//****************************************************************************************************
// Code generated by SFC Generator V1.13 on 13/03/19 15:52:14 by  David Paspa from File G:\Business\Synertec\MPI.SMS\automation\code\awlMaster\stencil\seq_hdr.awl
//****************************************************************************************************
//****************************************************************************************************

//================================ SEQ HEADER ================================//
//            Copyright 2018 Rieckermann Engineering Operations               //
//----------------------------------------------------------------------------//
// Title: PH_EMX1_SETUP_FILTER                                                       //
//                                                                            //
// Description:                                                               //
// Setup MMFLx for Filtration                                                        //
//                                                                            //
// // SFC Revision History:
// Rev By               Date        CC         Note
// 2.0 David Paspa      27-Nov-2018            Reboot for S7-1500
// 0.4 Khairul Basar    07-Sep-2009 CC-09/023  Prompt_filter is reset in Step2.
// 0.3 Khairul Basar    25-Aug-2009 CC-09/023  Change in Verific,& TRN code OR to AND
//                                             Change in the Last step.
// 0.2 Khairul Basar    18-Aug-2009            Added logic code
// 0.1 David Paspa      13-Jul-2009            SFC structural design                                                       //
//----------------------------------------------------------------------------//
// Sequencer Revision History:                                                //
// Rev By               Date        CC        Note                            //
// 2.0 David Paspa      05-Jan-2018 NA        Reboot for S7-1500.             //
// 1.6 Khairul Basar    19-Nov-2009 NA        Reset #sqSequencer.STEP.Active  //
//                                            when STEP Finished.             //
// 1.5 Khairul Basar    15-Oct-2009 NA        Placeholder inserted:           //
//                                            "udtSQ_PH";          //
// 1.4 Khairul Basar    06-Oct-2009 NA        R #PAUSE;                       //
// 1.3 Khairul Basar    30-Sep-2009 NA        SEQ_HDR change STEP-0 code      //
//                                            deleted.                        //
// 1.2 Khairul Basar    26-Sep-2009 NA        Refer R4.                       //
// 1.1 Khairul Basar    23-Sep-2009 NA        Refer R3.                       //
// 1.0 Khairul Basar    20-Sep-2009 NA        STEP.Finished flag reset by     //
//                                            JUMP_MAN.                       //
// 0.9 Khairul Basar    11-Sep-2009 NA        SQ_TIMER added as VAR, declared //
//                                            in SEQ_FTR.                     //
// 0.8 Khairul Basar    09-Sep-2009 NA        SqSequencer.Err_Fault is reset  //
//                                            on Stop cmd, Step-0 dead code   //
//                                            deleted from ACT & Verify.      //
//                                            STP_FTR Step_withErr flag       //
//                                            STEP_NUM place holder           //
//                                            configured.                     //
// 0.7 Khairul Basar    28-Aug-2009 NA        SQ_FINISHED OUT added again.    //
//                                            Deleted during major mod R3.    //
// 0.6 Khairul Basar    23-Aug-2009 NA        Refer R2.                       //
// 0.5 Khairul Basar    23-Aug-2009 NA        Refer R1.                       //
// 0.4 Khairul Basar    18-Aug-2009 NA        Reset Step done with/out error  //
//                                            bits using FC:RSET.             //
// 0.3 David Paspa      16-Aug-2009 NA        Added placeholders for header   //
//                                            name and version and revision   //
//                                            history.                        //
// 0.2 Khairul Basar    11-Aug-2009 NA        Retired external udt file for   //
//                                            Static type parameters. All     //
//                                            parameters now IN, OUT or       //
//                                            IN_OUT.                         //
// 0.1 Khairul Basar    12-Jun-2009 NA        Initial design.                 //
//----------------------------------------------------------------------------//
// R4:                                                                        //
// 1.If SQ not finished Resume command will start Step timer, and redo the    //
// last action, verify the feedback.                                          //
// 2."STEP.finished" flag is ANDed with "TRN_AND_JUMP" in the snippet file    //
// TRN_HDR.This is to avoid checking of transition logic if STEP is not       //
// finished yet.                                                              //
// 3.MDCH, Load & transfer typo corrected.                                    //
//                                                                            //
// R3:                                                                        //
// 1.SqStepTimer.IN is reset in STEP_FTR instead of resetting it in TRN_HDR.  //
// This is because TRN_HDTR is not included in the Last step and StepTimer    //
// must reset in the last step.                                               //
// 2.Reset all the timers when SQ stops.Reset done in SEQ_HDR.                //
// Also STEP-finished flag reset when SQ is OFF to                            //
// scan last step.                                                            //
//                                                                            //
// R2:                                                                        //
// 1.Any step error will send the Sequencer into Pause state.Code added in    //
// SEQ_HDR.Snippet Place holder for Bool-array 8 is   //
// deleted.                                                                   //
//                                                                            //
// R1:                                                                        //
// 1.sqStepTimer:All Verification Code must satisfy the condition finish step //
// action within STEP_DELAY time(40s).If step actions not finished within the //
// time period the error flag will raise High signal.Else timer will reset.   //
// 2.sqRunTimer Added therefore can be used as retentive & non retentive.     //
// 3.sqSequencer: This is re-structured UDT which is redefined the symbol     //
// names as well as it gives more clearity.                                   //
// 4.fcMODE and fcCMD functions are added to handle the mode & command        //
// independently regardless of other logic.Two separate UDT udtMODE & udt     //
// CMD assigned to Mode & command function respectively.                      //
// 5.MAN_JUMP programed for manual mode jump operation with or without        //
// Transition code satisfied.TRN_AND_JUMP & NO_VERIFC are the parameters      //
// which will define whether verification code & transition code need to be   //
// checked to perform jump operation.                                         //
// 6.Auto to Manual switchover will be bumpless & will not affect step        //
// operation.Manual to auto switchover can be used to resume Step action at   //
// defined.                                                                   //
// Step number entered in STEPNO_JUMP.                                        //
//                                                                            //
// Parameters:                                                                //
// INPUTS                                                                     //
// ======                                                                     //
// SQ_CMD          Sequence command input inherited from object block         //
//                 0: off/idle                                                //
//                 1: start/initiate                                          //
//                 2: pause                                                   //
//                 3: resume                                                  //
//                 4: reserved (not programmed)                               //
//                 5: reserved (not programmed)                               //
//                 6: abort/go to last step                                   //
//                 7: acknowledge error/fault                                 //
// SQ_MODE         Sequencer Auto/Manual input inherited from object block    //
//                 1: manual                                                  //
//                 2: auto                                                    //
//                                                                            //
// INPUT/OUTPUTS                                                              //
// =============                                                              //
// SQ_JUMP_MAN     Allows manual jumping from one step to the next step. The  //
//                 manual jump flag is ORed with the transition process       //
//                 condition and so can be used to bypass the condition if the//
//                 sequence will not progress.                                //
//                 This input can also be used to jump to any step even       //
//                 when no transition -> step linkage exists. This is only    //
//                 possible when the SQ_MODE is in manual and SQ is in the    //
//                 idle step. The step to jump to is specified in             //
//                 SQ_man_jump_to_step (not accesseble by this FB in/out      //
//                 interface but a separate DB memory location).              //
//                                                                            //
// OUTPUTS                                                                    //
// =======                                                                    //
// SQ_STATE        The calculated state of the sequence                       //
//                 0: off/idle                                                //
//                 1: start/initiated                                         //
//                 2: paused                                                  //
//                 3: resumed                                                 //
//                 4: reserved (wrong Mode)                                   //
//                 5: reserved (Wrong commad)                                 //
//                 6: aborted/go to last step                                 //
//                 7: acknowledged error/fault                                //
// CURSTEP         Current step being proccessed.                             //
// S_ACTIVE        If current step is active                                  //
// NXT_STEP        Next step to jump to if transition condition is true       //
// ERR_FAULT       True if any error/ or fault present                        //
// PAUSED          True if step is paused                                     //
// OFF_IDLE        Sequence is not running but ready for next SQ (in step=0)  //
//----------------------------------------------------------------------------//
// Define variables:                                                          //
//----------------------------------------------------------------------------//
FUNCTION_BLOCK "fbPH_EMX1_SETUP_FILTER"
TITLE = PH : EMX1_SETUP_FILTER
{ S7_Optimized_Access := 'TRUE' }
NAME : X1_FILT
AUTHOR : REO
VERSION : 2.0

VAR_IN_OUT
    _zsc_filter_state :INT ;	//MMFLx Filter connection sensor switch.

    _zsc_filter_cmd :INT ;	//FILTER connection command
    _zsc_cipsip_cmd :INT ;	//CIPSIP connection command


    dummy : bool;            // Dummy placeholder for call without comma
END_VAR

VAR
    smc : "udtModeCommandSFC";         // SFC mode and command
    sqStepTimer : "TON";
    sqRunTimer : "fbRunTimer";
    sqSequencer : "udtSFCSequence32";
    SQ_TIMER: "TON";
    SQ_TIMER2: "TON";
    SQ_TIMER3: "TON";
    sqSeqTimerStart : Bool;
    sqSeqTimerStart2 : Bool;
    sqSeqTimerStart3 : Bool;
    sqSeqTimerElapsed : Time;
    sqSeqTimerElapsed2 : Time;
    sqSeqTimerElapsed3 : Time;
    sqSeqTimerExpired : Bool;
    sqSeqTimerExpired2 : Bool;
    sqSeqTimerExpired3 : Bool;
    sqStepTimerElapsed : Time;
    sqStepTimerExpired : Bool;
    _log_msg_confirm_connect :BOOL ;	//PH_EMX1_SETUP_FILTER OPerator to confirm filters connected confirmed yes
    _log_msg_setup_filter_begin :BOOL ;	//PH_EMX1_SETUP_FILTER begin time
    _log_msg_setup_filter_end :BOOL ;	//PH_EMX1_SETUP_FILTER end time
    _prompt_connect_filter_confirm_yes :BOOL ;	//PH_EMX1_SETUP_FILTER operator to confirm filters connected confirmed yes
    _prompt_connect_filter :BOOL ;	//PH_EMX1_SETUP_FILTER Operator to confirm filters connected

END_VAR

BEGIN
NETWORK
TITLE =Call Mode checking function
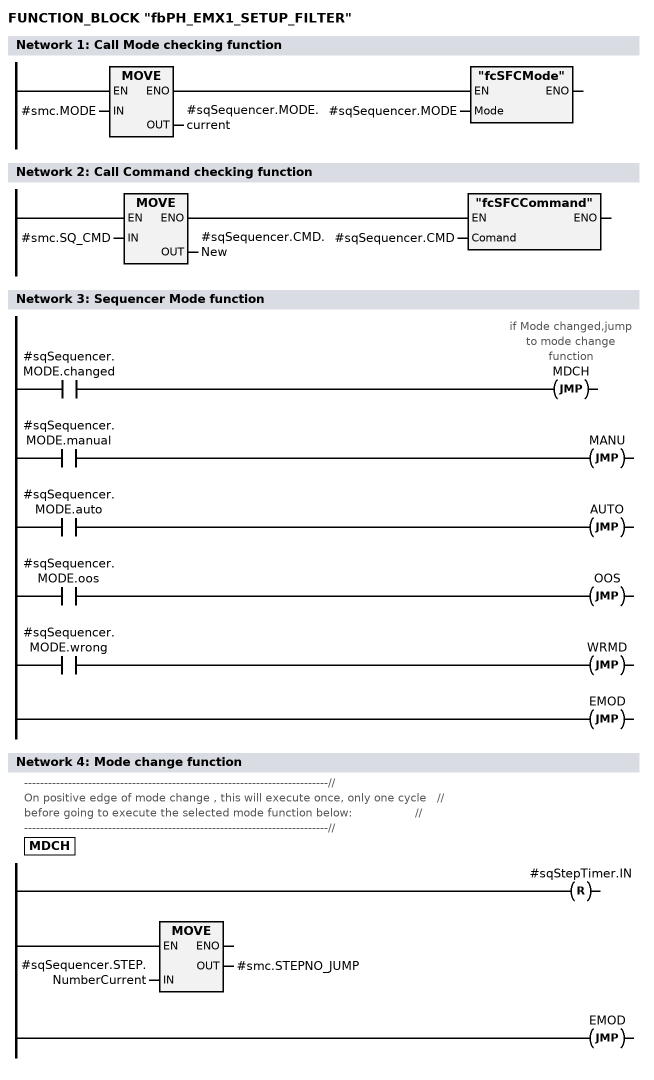
    L     #smc.MODE;
    T     #sqSequencer.MODE.current;
    CALL "fcSFCMode"
    (   Mode                 := #sqSequencer.MODE
    );

NETWORK
TITLE =Call Command checking function
    L     #smc.SQ_CMD;
    T     #sqSequencer.CMD.New;
    CALL "fcSFCCommand"
    (   Comand               := #sqSequencer.CMD
    );

NETWORK
TITLE =Sequencer Mode function

      A     #sqSequencer.MODE.changed;
      JC    MDCH; // if Mode changed,jump to mode change function
      A     #sqSequencer.MODE.manual;
      JC    MANU;
      A     #sqSequencer.MODE.auto;
      JC    AUTO;
      A     #sqSequencer.MODE.oos;
      JC    OOS;
      A     #sqSequencer.MODE.wrong;
      JC    WRMD;
      JU    EMOD;

NETWORK
TITLE =Mode change function
//----------------------------------------------------------------------------//
// On positive edge of mode change , this will execute once, only one cycle   //
// before going to execute the selected mode function below:                  //
//----------------------------------------------------------------------------//
MDCH: NOP   0;
      SET   ;
      R     #sqStepTimer.IN;
      L     #sqSequencer.STEP.NumberCurrent;
      T     #smc.STEPNO_JUMP;
      JU    EMOD;

NETWORK
TITLE =Manual Mode function
//----------------------------------------------------------------------------//
// #TRN_AND_JUMP=can set/reset                                                //
// #sqSequencer.STEP.JumpCtrl=Can set/reset by #MAN_JUMP                      //
// #NO_VERIFIC=Can set/ Reset                                                 //
//----------------------------------------------------------------------------//
MANU: NOP   0; //Manual mode selected



      A     #smc.MAN_JUMP;
      =     #sqSequencer.STEP.JumpCtrl;
      A     #smc.MAN_JUMP;
      JCN   EMOD;

      L     #smc.STEPNO_JUMP;
      T     #sqSequencer.STEP.NumberNext;
      T     #sqSequencer.STEP.NumberCurrent;
      R     #smc.MAN_JUMP; //Reset MAN_JUMP after loading user destination Step number
      R     #sqSequencer.STEP.Finished; //Reset finish flag, to execute next step action
      JU    EMOD;

NETWORK
TITLE =Auto Mode function
//----------------------------------------------------------------------------//
// #TRN_AND_JUMP=always set                                                   //
// #sqSequencer.STEP.JumpCtrl=Always set                                      //
// #NO_VERIFIC=Alwasy Reset                                                   //
//----------------------------------------------------------------------------//
AUTO: NOP   0; //Auto mode selected



      R     #smc.MAN_JUMP;
      S     #smc.TRN_AND_JUMP;
      R     #smc.NO_VERIFIC;
      S     #sqSequencer.STEP.JumpCtrl; //Always Set in auto mode

      L     #sqSequencer.STEP.NumberCurrent;
      T     #smc.STEPNO_JUMP;
      JU    EMOD;
NETWORK
TITLE =OOS mode function

OOS:  NOP   0; // Out of service
      JU    EMOD;
WRMD: NOP   0; //Wrong mode selected
      S     #sqSequencer.Error_Fault;
      L     "dbCONST".SEQ.STATE.WRMODE;
      T     #smc.SQ_STATE;

      JU    EMOD;

NETWORK
TITLE =Mode not changedd

      NOP   0;

NETWORK
TITLE =End Mode function

EMOD: NOP   0;

NETWORK
TITLE =An error will Pause the Sequencer,Operator must Resume SQ to run

      A     #sqSequencer.Error_Fault;
      AN    #sqSequencer.CMD.Changed;
      JC    PAUS;

NETWORK
TITLE =Command Action function

      A     #sqSequencer.CMD.Changed;
      JCN   CNCH; // if Command not changed,jump to end function
      R     #sqStepTimer.IN;

      A     #sqSequencer.CMD.Start;
      JC    STRT;

      A     #sqSequencer.CMD.Stop;
      JC    STOP;

      A     #sqSequencer.CMD.Pause;
      JC    PAUS;

      A     #sqSequencer.CMD.Resume;
      JC    RESM;

      A     #sqSequencer.CMD.Abort;
      JC    _abrt_begin;

      A     #sqSequencer.CMD.Ack;
      JC    ACKN;

      A     #sqSequencer.CMD.wrong;
      JC    WCMD;

      JU    ECMD; //Wrong command/not specified command
//End Comand function

NETWORK
TITLE =Comand -Start/Initiate action function

STRT: NOP   0;
      R     #smc.OFF_IDLE;
      R     #smc.ABORTED;
      R     #smc.PAUSED;
      R     #sqSequencer.STEP.Active;
      R     #sqSequencer.STEP.Finished;
      R     #sqSequencer.STEP.ActionFinished;
      R     #sqSequencer.STEP.Jump;
      R     #sqSequencer.STEP.TimerExpired;
      R     #sqSequencer.STEP.Error_Fault;
      R     #sqSequencer.STEP.ActionVerified;
      R     #sqStepTimer.IN;

//      S     #sqRunTimer.RESET;

//----------------------------------------------------------------------------//
// Load Initial step Number:                                                  //
//----------------------------------------------------------------------------//
      L     1;
      T     #sqSequencer.STEP.Initial;
      L     #sqSequencer.STEP.Initial;
      T     #sqSequencer.STEP.NumberCurrent;
      T     #sqSequencer.STEP.NumberNext;

      L     "dbCONST".SEQ.STATE.STARTED;
      T     #smc.SQ_STATE;

NETWORK
TITLE = Reset sequence Done bits
    //------------------------------------------------------------------------//
    // Reset Step done bits:                                                  //
    //------------------------------------------------------------------------//
    CALL FILL_BLK
    {value_type := 'Bool', count_type := 'UInt'}
    (   IN                   := 0 ,
        COUNT                := 32 ,
        OUT                  := #sqSequencer.STEP.Done[1]
    );

NETWORK
TITLE = Reset sequence Error bits
    //------------------------------------------------------------------------//
    // Reset Step error bits:                                                 //
    //------------------------------------------------------------------------//
    CALL FILL_BLK
    {value_type := 'Bool', count_type := 'UInt'}
    (   IN                   := 0 ,
        COUNT                := 32 ,
        OUT                  := #sqSequencer.STEP.WithError[1]
    );

    JU    ECMD; //End Function

NETWORK
TITLE =Comand -Stop action function

STOP: NOP   0;
      S     #smc.OFF_IDLE;
      R     #sqSequencer.STEP.Active;
      R     #sqSequencer.STEP.Finished;
      R     #sqSequencer.STEP.ActionFinished;
      R     #sqSequencer.STEP.Jump;
      R     #sqSequencer.STEP.TimerExpired;
      R     #sqSequencer.STEP.Error_Fault;
      R     #sqSequencer.Error_Fault;
      R     #sqSequencer.STEP.ActionVerified;
      R     #sqRunTimer.ENABLE;
      R     #sqStepTimer.IN;
      R     #sqSeqTimerStart;
      R     #sqSeqTimerStart2;
      R     #sqSeqTimerStart3;
      R     #smc.PAUSED;
      R     #smc.ABORTED;


//Go to last step
      L     4;
      T     #sqSequencer.FinalStep;
      T     #sqSequencer.STEP.NumberNext;

      JU    ECMD; //End Function

NETWORK
TITLE =Comand -Pause action function

PAUS: NOP   0;
      S     #smc.PAUSED;
      R     #smc.S_ACTIVE;
      S     #sqRunTimer.PAUSE;
      L     #sqSequencer.STEP.NumberCurrent;
      T     #smc.STEPNO_JUMP;
      L     "dbCONST".SEQ.STATE.PAUSED;
      T     #smc.SQ_STATE;

      JU    ECMD; //End Function

NETWORK
TITLE =Comand -Resume action function

RESM: NOP   0;
      R     #smc.PAUSED;
      R     #sqRunTimer.PAUSE;
      R     #sqStepTimer.IN; //Reset Step timer
      L     "dbCONST".SEQ.STATE.RESUMED;
      T     #smc.SQ_STATE;

      A     #smc.SQ_FINISHED;
      JC    ECMD;
      R     #sqSequencer.STEP.Active;
      R     #sqSequencer.STEP.Finished;
      R     #sqSequencer.STEP.ActionFinished;

      JU    ECMD; //End Function

NETWORK
TITLE =Comand -Abort action function

_abrt_begin: NOP   0;

      S     #smc.ABORTED;
      R     #sqSequencer.STEP.Active;
      R     #sqSequencer.STEP.Finished;
      R     #sqSequencer.STEP.ActionFinished;
      R     #sqSequencer.STEP.Jump;
      R     #sqSequencer.STEP.TimerExpired;
      R     #sqSequencer.STEP.Error_Fault;
      R     #sqSequencer.Error_Fault;
      R     #sqSequencer.STEP.ActionVerified;
      R     #sqRunTimer.ENABLE;
      R     #sqStepTimer.IN;
      R     #sqSeqTimerStart;
      R     #sqSeqTimerStart2;
      R     #sqSeqTimerStart3;
      R     #smc.PAUSED;
      R     #smc.OFF_IDLE;


//Go to last step
      L     4;
      T     #sqSequencer.FinalStep;
      T     #sqSequencer.STEP.NumberNext;

      JU    ECMD;

NETWORK
TITLE =Comand -Acknowledge action function

ACKN: NOP   0;
      R     #smc.ERR_FAULT;
      R     #sqSequencer.Error_Fault;
      L     "dbCONST".SEQ.STATE.ACKNOWLEDGED;
      T     #smc.SQ_STATE;

      JU    ECMD; //End Function

NETWORK
TITLE =Comand -wrong/unavailable

WCMD: NOP   0;

      S     #sqSequencer.Error_Fault;
      L     "dbCONST".SEQ.STATE.WRCMD;
      T     #smc.SQ_STATE;

      JU    ECMD;
NETWORK
TITLE =Comand -not changedd

CNCH: NOP   0; // Command not changed

NETWORK
TITLE =End command Function

ECMD: NOP   0;

NETWORK
TITLE =Sequencer Step Jump distrubution list
    //------------------------------------------------------------------------//
    // Sequencer step jump list. Load the step number to execute the step:    //
    //------------------------------------------------------------------------//
    L     #sqSequencer.STEP.NumberCurrent;
    JL    SQER; // If Sequencer Step number invalid or greater than available number of step
    JU    S000; // Exceptional Error Handling
    JU    S001; // STEP-001:
JU    S002; // STEP-002:
JU    S003; // STEP-003:
JU    S004; // STEP-004:


    //------------------------------------------------------------------------//
    // If Step number is Invalid or Out of Range:                             //
    //------------------------------------------------------------------------//
SQER: NOP   0;
    A     "alwaysLow";
    S     #sqSequencer.Error_Fault;
    JU    COMM; // Jump to Common Sequencer code handling function

NETWORK
TITLE =STEP0 STEP0 STEP0 STEP0 STEP0 STEP0 STEP0 STEP0 STEP0 STEP0 STEP
    //------------------------------------------------------------------------//
    // STEP0 STEP0 STEP0 STEP0 STEP0 STEP0 STEP0 STEP0 STEP0 STEP0 STEP0 STEP //
    // AUTOCODE   AUTOCODE   AUTOCODE   AUTOCODE   AUTOCODE   AUTOCODE   AUTO //
    // STEP0 STEP0 STEP0 STEP0 STEP0 STEP0 STEP0 STEP0 STEP0 STEP0 STEP0 STEP //
    //------------------------------------------------------------------------//

NETWORK
TITLE =S000: STEP0::If Paused exit

S000: NOP   0;
      JU    COMM;






NETWORK
TITLE =S001: STEP-01::PH_EMX1_SETUP_FILTER : SETUP CIPSIP begin.
    //================================ STEP HEADER ===========================//
    // STEP001 STEP001 STEP001 STEP001
    // AUTOCODE   AUTOCODE   AUTOCODE   AUTOCODE   AUTOCODE   AUTOCODE   AUTO //
    // STEP001 STEP001 STEP001 STEP001
    //------------------------------------------------------------------------//
    // Log SETUP FILTER begin time.
    //------------------------------------------------------------------------//
S001: NOP   0;

      SET;
      R     #sqSequencer.STEP.jumpDone[01];
      A     #sqSequencer.CMD.Pause; //If paused jump
      JC    COMM;

NETWORK
TITLE =S001:STEP-01:Begin Action

      A     #sqSequencer.STEP.Finished;
      JC    A001; // Exit Action code, Jump to A001 Transition code

      //----------------------------------------------------------------------//
      // Begin step Action:                                                   //
      //----------------------------------------------------------------------//
      A     #sqSequencer.STEP.Active;
      JC    L001; // Action number loaded, Jump to L001--Step Action List

      //----------------------------------------------------------------------//
      // Load Default/Initial Step action number:                             //
      //----------------------------------------------------------------------//
      S     #sqSequencer.STEP.Active;
      S     #sqStepTimer.IN;
      L     1; //First Action, Step must contain Minimum one action
      T     #sqSequencer.STEP.ActionNumber;

//----------------------------------------------------------------------------//
// Step action list.                                                          //
// aann=mini Action step number(aa) inside main step number(nn)               //
// First Action aa00, Second action ab00, Third ac00, etc.                    //
//----------------------------------------------------------------------------//
L001: NOP   0;

      L     #sqSequencer.STEP.ActionNumber;
      JL    r001; //Wrong Action number
      JU    _001; //Action error handling
       JU    aa01; //ACTION-01


//----------------------------------------------------------------------------//
// More step action in the list can be inserted here, upto ab is tested:      //
//----------------------------------------------------------------------------//
r001: NOP   0; //Wrong action number
      S     #sqSequencer.Error_Fault;
      JU    k001; //Exit
_001: NOP   0; // Action error handling
      JU    k001; // Exit






NETWORK
TITLE =S001:: STEP-001:: : ACTION CODE
    //================================ ACT HEADER ============================//
    // ACTION ACTION ACTION ACTION ACTION ACTION ACTION ACTION ACTION ACTION  //
    // AUTOCODE   AUTOCODE   AUTOCODE   AUTOCODE   AUTOCODE   AUTOCODE   AUTO //
    // ACTION ACTION ACTION ACTION ACTION ACTION ACTION ACTION ACTION ACTION  //
    //------------------------------------------------------------------------//
    // //Log SETUP FILTER begin time.
    aa01: NOP   0;

    //------------------------------------------------------------------------//
    // ACT ACT ACT ACT ACT ACT ACT ACT ACT ACT ACT ACT ACT ACT ACT ACT ACT    //
    //------------------------------------------------------------------------//
    //Log SETUP FILTER begin time.
SET;
S #_log_msg_setup_filter_begin;

// Send IN command to FILTER zsc.
L "dbCONST".BLK.ZSC2.CMD.IN;
T  #_zsc_filter_cmd;

// Send OUT command to CIPSIP zsc.
L "dbCONST".BLK.ZSC2.CMD.OUT;
T #_zsc_cipsip_cmd;

    //------------------------------------------------------------------------//
    // VERIFY  VERIFY VERIFY VERIFY VERIFY VERIFY VERIFY VERIFY VERIFY VERIFY //
    //------------------------------------------------------------------------//
    A "uncondJump";
    S     #sqSequencer.STEP.ActionVerified; //Action verified

    //------------------------------------------------------------------------//
    // Action done:                                                           //
    //------------------------------------------------------------------------//
    O     #sqSequencer.STEP.ActionVerified;
    O     #smc.NO_VERIFIC;       //No verification , bypass verification code
    S     #sqSequencer.STEP.ActionFinished;






    //============================= STEP FOOTER ==============================//
    // AUTOCODE   AUTOCODE   AUTOCODE   AUTOCODE   AUTOCODE   AUTOCODE   AUTO //
    // Get Ready after action finished:                                       //
    //------------------------------------------------------------------------//
    A     #sqSequencer.STEP.ActionFinished;
    JCN   k001;

    //------------------------------------------------------------------------//
    // Reset Action finished flag, ready for next step action:                //
    //------------------------------------------------------------------------//
    R     #sqSequencer.STEP.ActionVerified;
    R     #sqSequencer.STEP.ActionFinished;

    //------------------------------------------------------------------------//
    // If ALL actions are finished:                                           //
    //------------------------------------------------------------------------//
    SET   ;
    S     #sqSequencer.STEP.Finished;
    R     #sqSequencer.STEP.Active;
    S     #sqSequencer.STEP.Done[01];

    //------------------------------------------------------------------------//
    // End Step action(s):                                                    //
    //------------------------------------------------------------------------//
    JU    k001;

//----------------------------------------------------------------------------//
// Finished Step Action(s):                                                   //
//----------------------------------------------------------------------------//
k001: NOP   0;

    A     #sqStepTimerExpired;
    S     #sqSequencer.STEP.WithError[01]; // Step error flag
    S     #sqSequencer.Error_Fault;
    R     #sqStepTimer.IN;

NETWORK
TITLE =S001:STEP-001::Begin Transition
    //------------------------------------------------------------------------//
    // Begin the transition code:                                             //
    //------------------------------------------------------------------------//
    A001: NOP   0;
    R     #sqStepTimer.IN;






    //============================= TRAN HEADER ==============================//
    // AUTOCODE   AUTOCODE   AUTOCODE   AUTOCODE   AUTOCODE   AUTOCODE   AUTO //
    // Bypass transition if manual jump:                                      //
    //------------------------------------------------------------------------//
    A     #sqSequencer.STEP.Finished;
    A     #smc.TRN_AND_JUMP;     //Manual jump is set Transition as bypassed
    JCN   COMM;              //exit

NETWORK
TITLE =S001::STEP 001:TRAN 001: Unconditional Jump
//----------------------------------------------------------------------------//
// TRAN   TRAN   TRAN   TRAN   TRAN   TRAN   TRAN   TRAN   TRAN   TRAN   TRAN //
// TRAN   TRAN   TRAN   TRAN   TRAN   TRAN   TRAN   TRAN   TRAN   TRAN   TRAN //
//----------------------------------------------------------------------------//
// Jump
//----------------------------------------------------------------------------//
// CONDITION   CONDITION   CONDITION   CONDITION   CONDITION   CONDITION   CO //
// CONDITION   CONDITION   CONDITION   CONDITION   CONDITION   CONDITION   CO //
//----------------------------------------------------------------------------//
A "uncondJump";






    //============================= TRAN FOOTER ==============================//
    // Transition jump control:                                               //
    //------------------------------------------------------------------------//
    A     #sqSequencer.STEP.JumpCtrl;
    S     #sqSequencer.STEP.Jump;
    S     #sqSequencer.STEP.jumpDone[01];

NETWORK
TITLE =S001:t001::TRANS-v: EXIT TRANSITION AND READY THE NEXT STEP
    //------------------------------------------------------------------------//
    // Check the jump flag and jump to the next step if the transition        //
    // condition is true and has set the jump flag:                           //
    //------------------------------------------------------------------------//
    A     #sqSequencer.STEP.Jump;
    JCN   x001;

    R     #sqSequencer.STEP.Jump;
    R     #sqSequencer.STEP.Finished;

    L     02;     // Load next STEPNO to jump to if transition satisfied
    T     #sqSequencer.STEP.NumberNext; //Next Step02.

    JU    COMM;              // Transition satisfied, Exit, go to next step
x001: NOP   0;






NETWORK
TITLE =S001::STEP-001:EXIT TRANSITION:
    //========================== STEP TRANSFER ===============================//
    // Jump to the common step progression code:                              //
    //------------------------------------------------------------------------//
    JU    COMM;






NETWORK
TITLE =S002: STEP-02::PH_EMX1_SETUP_FILTER : Prompt operator to connect jumpers
    //================================ STEP HEADER ===========================//
    // STEP002 STEP002 STEP002 STEP002
    // AUTOCODE   AUTOCODE   AUTOCODE   AUTOCODE   AUTOCODE   AUTOCODE   AUTO //
    // STEP002 STEP002 STEP002 STEP002
    //------------------------------------------------------------------------//
    // Prompt operator to connect jumpers on FP11:
    // M1 to Pre-Filter: ZSCx113
    //------------------------------------------------------------------------//
S002: NOP   0;

      SET;
      R     #sqSequencer.STEP.jumpDone[02];
      A     #sqSequencer.CMD.Pause; //If paused jump
      JC    COMM;

NETWORK
TITLE =S002:STEP-02:Begin Action

      A     #sqSequencer.STEP.Finished;
      JC    A002; // Exit Action code, Jump to A002 Transition code

      //----------------------------------------------------------------------//
      // Begin step Action:                                                   //
      //----------------------------------------------------------------------//
      A     #sqSequencer.STEP.Active;
      JC    L002; // Action number loaded, Jump to L002--Step Action List

      //----------------------------------------------------------------------//
      // Load Default/Initial Step action number:                             //
      //----------------------------------------------------------------------//
      S     #sqSequencer.STEP.Active;
      S     #sqStepTimer.IN;
      L     1; //First Action, Step must contain Minimum one action
      T     #sqSequencer.STEP.ActionNumber;

//----------------------------------------------------------------------------//
// Step action list.                                                          //
// aann=mini Action step number(aa) inside main step number(nn)               //
// First Action aa00, Second action ab00, Third ac00, etc.                    //
//----------------------------------------------------------------------------//
L002: NOP   0;

      L     #sqSequencer.STEP.ActionNumber;
      JL    r002; //Wrong Action number
      JU    _002; //Action error handling
       JU    aa02; //ACTION-01


//----------------------------------------------------------------------------//
// More step action in the list can be inserted here, upto ab is tested:      //
//----------------------------------------------------------------------------//
r002: NOP   0; //Wrong action number
      S     #sqSequencer.Error_Fault;
      JU    k002; //Exit
_002: NOP   0; // Action error handling
      JU    k002; // Exit






NETWORK
TITLE =S002:: STEP-002:: : ACTION CODE
    //================================ ACT HEADER ============================//
    // ACTION ACTION ACTION ACTION ACTION ACTION ACTION ACTION ACTION ACTION  //
    // AUTOCODE   AUTOCODE   AUTOCODE   AUTOCODE   AUTOCODE   AUTOCODE   AUTO //
    // ACTION ACTION ACTION ACTION ACTION ACTION ACTION ACTION ACTION ACTION  //
    //------------------------------------------------------------------------//
    // //Prompt operator to connect the filter
    aa02: NOP   0;

    //------------------------------------------------------------------------//
    // ACT ACT ACT ACT ACT ACT ACT ACT ACT ACT ACT ACT ACT ACT ACT ACT ACT    //
    //------------------------------------------------------------------------//
    //Prompt to connect filter.
SET;
S #_prompt_connect_filter;

    //------------------------------------------------------------------------//
    // VERIFY  VERIFY VERIFY VERIFY VERIFY VERIFY VERIFY VERIFY VERIFY VERIFY //
    //------------------------------------------------------------------------//
    A "uncondJump";
    S     #sqSequencer.STEP.ActionVerified; //Action verified

    //------------------------------------------------------------------------//
    // Action done:                                                           //
    //------------------------------------------------------------------------//
    O     #sqSequencer.STEP.ActionVerified;
    O     #smc.NO_VERIFIC;       //No verification , bypass verification code
    S     #sqSequencer.STEP.ActionFinished;






    //============================= STEP FOOTER ==============================//
    // AUTOCODE   AUTOCODE   AUTOCODE   AUTOCODE   AUTOCODE   AUTOCODE   AUTO //
    // Get Ready after action finished:                                       //
    //------------------------------------------------------------------------//
    A     #sqSequencer.STEP.ActionFinished;
    JCN   k002;

    //------------------------------------------------------------------------//
    // Reset Action finished flag, ready for next step action:                //
    //------------------------------------------------------------------------//
    R     #sqSequencer.STEP.ActionVerified;
    R     #sqSequencer.STEP.ActionFinished;

    //------------------------------------------------------------------------//
    // If ALL actions are finished:                                           //
    //------------------------------------------------------------------------//
    SET   ;
    S     #sqSequencer.STEP.Finished;
    R     #sqSequencer.STEP.Active;
    S     #sqSequencer.STEP.Done[02];

    //------------------------------------------------------------------------//
    // End Step action(s):                                                    //
    //------------------------------------------------------------------------//
    JU    k002;

//----------------------------------------------------------------------------//
// Finished Step Action(s):                                                   //
//----------------------------------------------------------------------------//
k002: NOP   0;

    A     #sqStepTimerExpired;
    S     #sqSequencer.STEP.WithError[02]; // Step error flag
    S     #sqSequencer.Error_Fault;
    R     #sqStepTimer.IN;

NETWORK
TITLE =S002:STEP-002::Begin Transition
    //------------------------------------------------------------------------//
    // Begin the transition code:                                             //
    //------------------------------------------------------------------------//
    A002: NOP   0;
    R     #sqStepTimer.IN;






    //============================= TRAN HEADER ==============================//
    // AUTOCODE   AUTOCODE   AUTOCODE   AUTOCODE   AUTOCODE   AUTOCODE   AUTO //
    // Bypass transition if manual jump:                                      //
    //------------------------------------------------------------------------//
    A     #sqSequencer.STEP.Finished;
    A     #smc.TRN_AND_JUMP;     //Manual jump is set Transition as bypassed
    JCN   COMM;              //exit

NETWORK
TITLE =S002::STEP 002:TRAN 002: Operator confirmation
//----------------------------------------------------------------------------//
// TRAN   TRAN   TRAN   TRAN   TRAN   TRAN   TRAN   TRAN   TRAN   TRAN   TRAN //
// TRAN   TRAN   TRAN   TRAN   TRAN   TRAN   TRAN   TRAN   TRAN   TRAN   TRAN //
//----------------------------------------------------------------------------//
// Wait for operator to confirm connections has been made.
//----------------------------------------------------------------------------//
// CONDITION   CONDITION   CONDITION   CONDITION   CONDITION   CONDITION   CO //
// CONDITION   CONDITION   CONDITION   CONDITION   CONDITION   CONDITION   CO //
//----------------------------------------------------------------------------//
A #_prompt_connect_filter_confirm_yes;






    //============================= TRAN FOOTER ==============================//
    // Transition jump control:                                               //
    //------------------------------------------------------------------------//
    A     #sqSequencer.STEP.JumpCtrl;
    S     #sqSequencer.STEP.Jump;
    S     #sqSequencer.STEP.jumpDone[02];

NETWORK
TITLE =S002:t002::TRANS-v: EXIT TRANSITION AND READY THE NEXT STEP
    //------------------------------------------------------------------------//
    // Check the jump flag and jump to the next step if the transition        //
    // condition is true and has set the jump flag:                           //
    //------------------------------------------------------------------------//
    A     #sqSequencer.STEP.Jump;
    JCN   x002;

    R     #sqSequencer.STEP.Jump;
    R     #sqSequencer.STEP.Finished;

    L     03;     // Load next STEPNO to jump to if transition satisfied
    T     #sqSequencer.STEP.NumberNext; //Next Step03.

    JU    COMM;              // Transition satisfied, Exit, go to next step
x002: NOP   0;






NETWORK
TITLE =S002::STEP-002:EXIT TRANSITION:
    //========================== STEP TRANSFER ===============================//
    // Jump to the common step progression code:                              //
    //------------------------------------------------------------------------//
    JU    COMM;






NETWORK
TITLE =S003: STEP-03::PH_EMX1_SETUP_FILTER : Check connection
    //================================ STEP HEADER ===========================//
    // STEP003 STEP003 STEP003 STEP003
    // AUTOCODE   AUTOCODE   AUTOCODE   AUTOCODE   AUTOCODE   AUTOCODE   AUTO //
    // STEP003 STEP003 STEP003 STEP003
    //------------------------------------------------------------------------//
    // Log operator confirmation and continue to check connection.
    //------------------------------------------------------------------------//
S003: NOP   0;

      SET;
      R     #sqSequencer.STEP.jumpDone[03];
      A     #sqSequencer.CMD.Pause; //If paused jump
      JC    COMM;

NETWORK
TITLE =S003:STEP-03:Begin Action

      A     #sqSequencer.STEP.Finished;
      JC    A003; // Exit Action code, Jump to A003 Transition code

      //----------------------------------------------------------------------//
      // Begin step Action:                                                   //
      //----------------------------------------------------------------------//
      A     #sqSequencer.STEP.Active;
      JC    L003; // Action number loaded, Jump to L003--Step Action List

      //----------------------------------------------------------------------//
      // Load Default/Initial Step action number:                             //
      //----------------------------------------------------------------------//
      S     #sqSequencer.STEP.Active;
      S     #sqStepTimer.IN;
      L     1; //First Action, Step must contain Minimum one action
      T     #sqSequencer.STEP.ActionNumber;

//----------------------------------------------------------------------------//
// Step action list.                                                          //
// aann=mini Action step number(aa) inside main step number(nn)               //
// First Action aa00, Second action ab00, Third ac00, etc.                    //
//----------------------------------------------------------------------------//
L003: NOP   0;

      L     #sqSequencer.STEP.ActionNumber;
      JL    r003; //Wrong Action number
      JU    _003; //Action error handling
       JU    aa03; //ACTION-01


//----------------------------------------------------------------------------//
// More step action in the list can be inserted here, upto ab is tested:      //
//----------------------------------------------------------------------------//
r003: NOP   0; //Wrong action number
      S     #sqSequencer.Error_Fault;
      JU    k003; //Exit
_003: NOP   0; // Action error handling
      JU    k003; // Exit






NETWORK
TITLE =S003:: STEP-003:: : ACTION CODE
    //================================ ACT HEADER ============================//
    // ACTION ACTION ACTION ACTION ACTION ACTION ACTION ACTION ACTION ACTION  //
    // AUTOCODE   AUTOCODE   AUTOCODE   AUTOCODE   AUTOCODE   AUTOCODE   AUTO //
    // ACTION ACTION ACTION ACTION ACTION ACTION ACTION ACTION ACTION ACTION  //
    //------------------------------------------------------------------------//
    // //Log operator confirmation and continue to check connection.
    aa03: NOP   0;

    //------------------------------------------------------------------------//
    // ACT ACT ACT ACT ACT ACT ACT ACT ACT ACT ACT ACT ACT ACT ACT ACT ACT    //
    //------------------------------------------------------------------------//
    SET;
S #_log_msg_confirm_connect;

    //------------------------------------------------------------------------//
    // VERIFY  VERIFY VERIFY VERIFY VERIFY VERIFY VERIFY VERIFY VERIFY VERIFY //
    //------------------------------------------------------------------------//
    A "uncondJump";
    S     #sqSequencer.STEP.ActionVerified; //Action verified

    //------------------------------------------------------------------------//
    // Action done:                                                           //
    //------------------------------------------------------------------------//
    O     #sqSequencer.STEP.ActionVerified;
    O     #smc.NO_VERIFIC;       //No verification , bypass verification code
    S     #sqSequencer.STEP.ActionFinished;






    //============================= STEP FOOTER ==============================//
    // AUTOCODE   AUTOCODE   AUTOCODE   AUTOCODE   AUTOCODE   AUTOCODE   AUTO //
    // Get Ready after action finished:                                       //
    //------------------------------------------------------------------------//
    A     #sqSequencer.STEP.ActionFinished;
    JCN   k003;

    //------------------------------------------------------------------------//
    // Reset Action finished flag, ready for next step action:                //
    //------------------------------------------------------------------------//
    R     #sqSequencer.STEP.ActionVerified;
    R     #sqSequencer.STEP.ActionFinished;

    //------------------------------------------------------------------------//
    // If ALL actions are finished:                                           //
    //------------------------------------------------------------------------//
    SET   ;
    S     #sqSequencer.STEP.Finished;
    R     #sqSequencer.STEP.Active;
    S     #sqSequencer.STEP.Done[03];

    //------------------------------------------------------------------------//
    // End Step action(s):                                                    //
    //------------------------------------------------------------------------//
    JU    k003;

//----------------------------------------------------------------------------//
// Finished Step Action(s):                                                   //
//----------------------------------------------------------------------------//
k003: NOP   0;

    A     #sqStepTimerExpired;
    S     #sqSequencer.STEP.WithError[03]; // Step error flag
    S     #sqSequencer.Error_Fault;
    R     #sqStepTimer.IN;

NETWORK
TITLE =S003:STEP-003::Begin Transition
    //------------------------------------------------------------------------//
    // Begin the transition code:                                             //
    //------------------------------------------------------------------------//
    A003: NOP   0;
    R     #sqStepTimer.IN;






    //============================= TRAN HEADER ==============================//
    // AUTOCODE   AUTOCODE   AUTOCODE   AUTOCODE   AUTOCODE   AUTOCODE   AUTO //
    // Bypass transition if manual jump:                                      //
    //------------------------------------------------------------------------//
    A     #sqSequencer.STEP.Finished;
    A     #smc.TRN_AND_JUMP;     //Manual jump is set Transition as bypassed
    JCN   COMM;              //exit

NETWORK
TITLE =S003::STEP 003:TRAN 003: Connection correctly inserted
//----------------------------------------------------------------------------//
// TRAN   TRAN   TRAN   TRAN   TRAN   TRAN   TRAN   TRAN   TRAN   TRAN   TRAN //
// TRAN   TRAN   TRAN   TRAN   TRAN   TRAN   TRAN   TRAN   TRAN   TRAN   TRAN //
//----------------------------------------------------------------------------//
// Jump if correct switch ZSCx113 connected
//----------------------------------------------------------------------------//
// CONDITION   CONDITION   CONDITION   CONDITION   CONDITION   CONDITION   CO //
// CONDITION   CONDITION   CONDITION   CONDITION   CONDITION   CONDITION   CO //
//----------------------------------------------------------------------------//
//Verify the correct switch connected.
A(;
L #_zsc_filter_state;
L "dbCONST".BLK.ZSC2.STATE.IN;
==I ;
);






    //============================= TRAN FOOTER ==============================//
    // Transition jump control:                                               //
    //------------------------------------------------------------------------//
    A     #sqSequencer.STEP.JumpCtrl;
    S     #sqSequencer.STEP.Jump;
    S     #sqSequencer.STEP.jumpDone[03];

NETWORK
TITLE =S003:t003::TRANS-v: EXIT TRANSITION AND READY THE NEXT STEP
    //------------------------------------------------------------------------//
    // Check the jump flag and jump to the next step if the transition        //
    // condition is true and has set the jump flag:                           //
    //------------------------------------------------------------------------//
    A     #sqSequencer.STEP.Jump;
    JCN   x003;

    R     #sqSequencer.STEP.Jump;
    R     #sqSequencer.STEP.Finished;

    L     04;     // Load next STEPNO to jump to if transition satisfied
    T     #sqSequencer.STEP.NumberNext; //Next Step04.

    JU    COMM;              // Transition satisfied, Exit, go to next step
x003: NOP   0;






    //============================= TRAN HEADER ==============================//
    // AUTOCODE   AUTOCODE   AUTOCODE   AUTOCODE   AUTOCODE   AUTOCODE   AUTO //
    // Bypass transition if manual jump:                                      //
    //------------------------------------------------------------------------//
    A     #sqSequencer.STEP.Finished;
    A     #smc.TRN_AND_JUMP;     //Manual jump is set Transition as bypassed
    JCN   COMM;              //exit

NETWORK
TITLE =S003::STEP 003:TRAN 004: Operator not setup correctly
//----------------------------------------------------------------------------//
// TRAN   TRAN   TRAN   TRAN   TRAN   TRAN   TRAN   TRAN   TRAN   TRAN   TRAN //
// TRAN   TRAN   TRAN   TRAN   TRAN   TRAN   TRAN   TRAN   TRAN   TRAN   TRAN //
//----------------------------------------------------------------------------//
// Jump unconditionally, the connections are not made correctly
//----------------------------------------------------------------------------//
// CONDITION   CONDITION   CONDITION   CONDITION   CONDITION   CONDITION   CO //
// CONDITION   CONDITION   CONDITION   CONDITION   CONDITION   CONDITION   CO //
//----------------------------------------------------------------------------//
A "uncondJump";






    //============================= TRAN FOOTER ==============================//
    // Transition jump control:                                               //
    //------------------------------------------------------------------------//
    A     #sqSequencer.STEP.JumpCtrl;
    S     #sqSequencer.STEP.Jump;
    S     #sqSequencer.STEP.jumpDone[03];

NETWORK
TITLE =S003:t004::TRANS-v: EXIT TRANSITION AND READY THE NEXT STEP
    //------------------------------------------------------------------------//
    // Check the jump flag and jump to the next step if the transition        //
    // condition is true and has set the jump flag:                           //
    //------------------------------------------------------------------------//
    A     #sqSequencer.STEP.Jump;
    JCN   x004;

    R     #sqSequencer.STEP.Jump;
    R     #sqSequencer.STEP.Finished;

    L     02;     // Load next STEPNO to jump to if transition satisfied
    T     #sqSequencer.STEP.NumberNext; //Next Step02.

    JU    COMM;              // Transition satisfied, Exit, go to next step
x004: NOP   0;






NETWORK
TITLE =S003::STEP-003:EXIT TRANSITION:
    //========================== STEP TRANSFER ===============================//
    // Jump to the common step progression code:                              //
    //------------------------------------------------------------------------//
    JU    COMM;






NETWORK
TITLE =S004: STEP-04::PH_EMX1_SETUP_FILTER : Last Step
    //================================ STEP HEADER ===========================//
    // STEP004 STEP004 STEP004 STEP004
    // AUTOCODE   AUTOCODE   AUTOCODE   AUTOCODE   AUTOCODE   AUTOCODE   AUTO //
    // STEP004 STEP004 STEP004 STEP004
    //------------------------------------------------------------------------//
    // Log SETUP FILTER operation end time.
    //------------------------------------------------------------------------//
S004: NOP   0;

      SET;
      R     #sqSequencer.STEP.jumpDone[04];
      A     #sqSequencer.CMD.Pause; //If paused jump
      JC    COMM;

NETWORK
TITLE =S004:STEP-04:Begin Action

      A     #sqSequencer.STEP.Finished;
      JC    A004; // Exit Action code, Jump to A004 Transition code

      //----------------------------------------------------------------------//
      // Begin step Action:                                                   //
      //----------------------------------------------------------------------//
      A     #sqSequencer.STEP.Active;
      JC    L004; // Action number loaded, Jump to L004--Step Action List

      //----------------------------------------------------------------------//
      // Load Default/Initial Step action number:                             //
      //----------------------------------------------------------------------//
      S     #sqSequencer.STEP.Active;
      S     #sqStepTimer.IN;
      L     1; //First Action, Step must contain Minimum one action
      T     #sqSequencer.STEP.ActionNumber;

//----------------------------------------------------------------------------//
// Step action list.                                                          //
// aann=mini Action step number(aa) inside main step number(nn)               //
// First Action aa00, Second action ab00, Third ac00, etc.                    //
//----------------------------------------------------------------------------//
L004: NOP   0;

      L     #sqSequencer.STEP.ActionNumber;
      JL    r004; //Wrong Action number
      JU    _004; //Action error handling
       JU    aa04; //ACTION-01


//----------------------------------------------------------------------------//
// More step action in the list can be inserted here, upto ab is tested:      //
//----------------------------------------------------------------------------//
r004: NOP   0; //Wrong action number
      S     #sqSequencer.Error_Fault;
      JU    k004; //Exit
_004: NOP   0; // Action error handling
      JU    k004; // Exit






NETWORK
TITLE =S004:: STEP-004:: : ACTION CODE
    //================================ ACT HEADER ============================//
    // ACTION ACTION ACTION ACTION ACTION ACTION ACTION ACTION ACTION ACTION  //
    // AUTOCODE   AUTOCODE   AUTOCODE   AUTOCODE   AUTOCODE   AUTOCODE   AUTO //
    // ACTION ACTION ACTION ACTION ACTION ACTION ACTION ACTION ACTION ACTION  //
    //------------------------------------------------------------------------//
    // //Log SETUP FILTER operation end time.
    aa04: NOP   0;

    //------------------------------------------------------------------------//
    // ACT ACT ACT ACT ACT ACT ACT ACT ACT ACT ACT ACT ACT ACT ACT ACT ACT    //
    //------------------------------------------------------------------------//
    //Log SETUP FILTER operation end time.
SET;
S #_log_msg_setup_filter_end;

    //------------------------------------------------------------------------//
    // VERIFY  VERIFY VERIFY VERIFY VERIFY VERIFY VERIFY VERIFY VERIFY VERIFY //
    //------------------------------------------------------------------------//
    A "uncondJump";
    S     #sqSequencer.STEP.ActionVerified; //Action verified

    //------------------------------------------------------------------------//
    // Action done:                                                           //
    //------------------------------------------------------------------------//
    O     #sqSequencer.STEP.ActionVerified;
    O     #smc.NO_VERIFIC;       //No verification , bypass verification code
    S     #sqSequencer.STEP.ActionFinished;






    //============================= STEP FOOTER ==============================//
    // AUTOCODE   AUTOCODE   AUTOCODE   AUTOCODE   AUTOCODE   AUTOCODE   AUTO //
    // Get Ready after action finished:                                       //
    //------------------------------------------------------------------------//
    A     #sqSequencer.STEP.ActionFinished;
    JCN   k004;

    //------------------------------------------------------------------------//
    // Reset Action finished flag, ready for next step action:                //
    //------------------------------------------------------------------------//
    R     #sqSequencer.STEP.ActionVerified;
    R     #sqSequencer.STEP.ActionFinished;

    //------------------------------------------------------------------------//
    // If ALL actions are finished:                                           //
    //------------------------------------------------------------------------//
    SET   ;
    S     #sqSequencer.STEP.Finished;
    R     #sqSequencer.STEP.Active;
    S     #sqSequencer.STEP.Done[04];

    //------------------------------------------------------------------------//
    // End Step action(s):                                                    //
    //------------------------------------------------------------------------//
    JU    k004;

//----------------------------------------------------------------------------//
// Finished Step Action(s):                                                   //
//----------------------------------------------------------------------------//
k004: NOP   0;

    A     #sqStepTimerExpired;
    S     #sqSequencer.STEP.WithError[04]; // Step error flag
    S     #sqSequencer.Error_Fault;
    R     #sqStepTimer.IN;

NETWORK
TITLE =S004:STEP-004::Begin Transition
    //------------------------------------------------------------------------//
    // Begin the transition code:                                             //
    //------------------------------------------------------------------------//
    A004: NOP   0;
    R     #sqStepTimer.IN;






NETWORK
TITLE =S004::STEP-004:EXIT TRANSITION:
    //========================== STEP TRANSFER ===============================//
    // Jump to the common step progression code:                              //
    //------------------------------------------------------------------------//
    JU    COMM;






NETWORK
TITLE =Sequencer Common Code, Execute in Each Scan
    //============================ SEQ FOOTER ================================//
    // AUTOCODE   AUTOCODE   AUTOCODE   AUTOCODE   AUTOCODE   AUTOCODE   AUTO //
    // Common code to execute each scan:                                      //
    //------------------------------------------------------------------------//
    COMM: NOP   0;

NETWORK
TITLE =Retentive/Non Retentive Selectable Run timer
    CALL #sqRunTimer (
        TIME_H               := #sqRunTimer.TIME_H,
        TIME_M               := #sqRunTimer.TIME_M,
        TIME_S               := #sqRunTimer.TIME_S,
        ENABLE               := #sqRunTimer.ENABLE,
        RESET                := #sqRunTimer.RESET,
        PAUSE                := #sqRunTimer.PAUSE,
        NON_RET              := #sqRunTimer.NON_RET,
        RMNG_H               := #sqRunTimer.RMNG_H,
        RMNG_M               := #sqRunTimer.RMNG_M,
        RMNG_S               := #sqRunTimer.RMNG_S,
        TIME_EXPIRED         := #sqRunTimer.TIME_EXPIRED,
        TMR_RUNNG            := #sqRunTimer.TMR_RUNNG
    );

NETWORK
TITLE =Sequencer Step Timer
    CALL #sqStepTimer (
        IN                   := #sqStepTimer.IN,
        PT                   := "dbCONST".SEQ.STEP_TIME,
        Q                    := #sqStepTimerExpired,
        ET                   := #sqStepTimerElapsed
    );

NETWORK
TITLE =Sequencer Timer
    CALL #SQ_TIMER (
        IN                   := #sqSeqTimerStart,
        PT                   := #SQ_TIMER.PT,
        Q                    := #sqSeqTimerExpired,
        ET                   := #sqSeqTimerElapsed
    );

    CALL #SQ_TIMER2 (
        IN                   := #sqSeqTimerStart2,
        PT                   := #SQ_TIMER2.PT,
        Q                    := #sqSeqTimerExpired2,
        ET                   := #sqSeqTimerElapsed2
    );

NETWORK
TITLE =Sequencer Timer
    CALL #SQ_TIMER3 (
        IN                   := #sqSeqTimerStart3,
        PT                   := #SQ_TIMER3.PT,
        Q                    := #sqSeqTimerExpired3,
        ET                   := #sqSeqTimerElapsed3
    );

NETWORK
TITLE =General Assignments

    L     #sqSequencer.STEP.NumberNext;
    T     #smc.NXT_STEP;
    T     #sqSequencer.STEP.NumberCurrent;
    T     #smc.CURSTEP;

    A     #sqSequencer.STEP.Active;
    =     #smc.S_ACTIVE;

    A     #sqSequencer.Error_Fault;
    =     #smc.ERR_FAULT;

NETWORK
TITLE = Stop command completion
    A    #smc.OFF_IDLE;
    A    #sqSequencer.STEP.Done[4];
    AN   #sqSequencer.STEP.WithError[4];
    JCN NotStopCmd;
    R    #smc.PAUSED;
    R    #sqSequencer.STEP.Error_Fault;
    R    #sqSequencer.Error_Fault;
    L    "dbCONST".SEQ.STATE.OFF_IDLE;
    T    #smc.SQ_STATE;
NotStopCmd:   NOP 0;

    A    #smc.OFF_IDLE;
    AN    #sqSequencer.STEP.Done[4];
    AN    #sqSequencer.STEP.WithError[4];
    JCN   _stopAction;
    R     #sqSequencer.STEP.Finished;
    R     #smc.PAUSED;
    R     #sqSequencer.STEP.Error_Fault;
    R     #sqSequencer.Error_Fault;
_stopAction:   NOP 0;

NETWORK
TITLE =Sequencer Finished

    AN    #smc.OFF_IDLE;
    AN    #smc.PAUSED;
    A     #sqSequencer.STEP.Done[4];
    =     #sqSequencer.Finished;
    =     #smc.SQ_FINISHED;
    JCN   fnsd;
    L     "dbCONST".SEQ.STATE.COMPLETED;
    T     #smc.SQ_STATE;
    R     #smc.PAUSED;
    R     #sqSequencer.STEP.Error_Fault;
    R     #sqSequencer.Error_Fault;
fnsd: NOP   0;

    //------------------------------------------------------------------------//
    // Reset Finished flag if SQ OFF for Last step to scan:                   //
    //------------------------------------------------------------------------//
    A     #smc.ABORTED;
    AN    #sqSequencer.STEP.Done[4];
    AN    #sqSequencer.STEP.WithError[4];
    JCN   _abrt_end;
    R     #sqSequencer.STEP.Finished;
    R     #smc.PAUSED;
    R     #sqSequencer.STEP.Error_Fault;
    R     #sqSequencer.Error_Fault;
    L     "dbCONST".SEQ.STATE.ABORTED;
    T     #smc.SQ_STATE;
_abrt_end: NOP   0;

    //------------------------------------------------------------------------//
    // Visio Common Code Begin:                                               //
    //------------------------------------------------------------------------//


//----------------------------------------------------------------------------//
// End of Sequencer:                                                          //
//----------------------------------------------------------------------------//
END_FUNCTION_BLOCK

